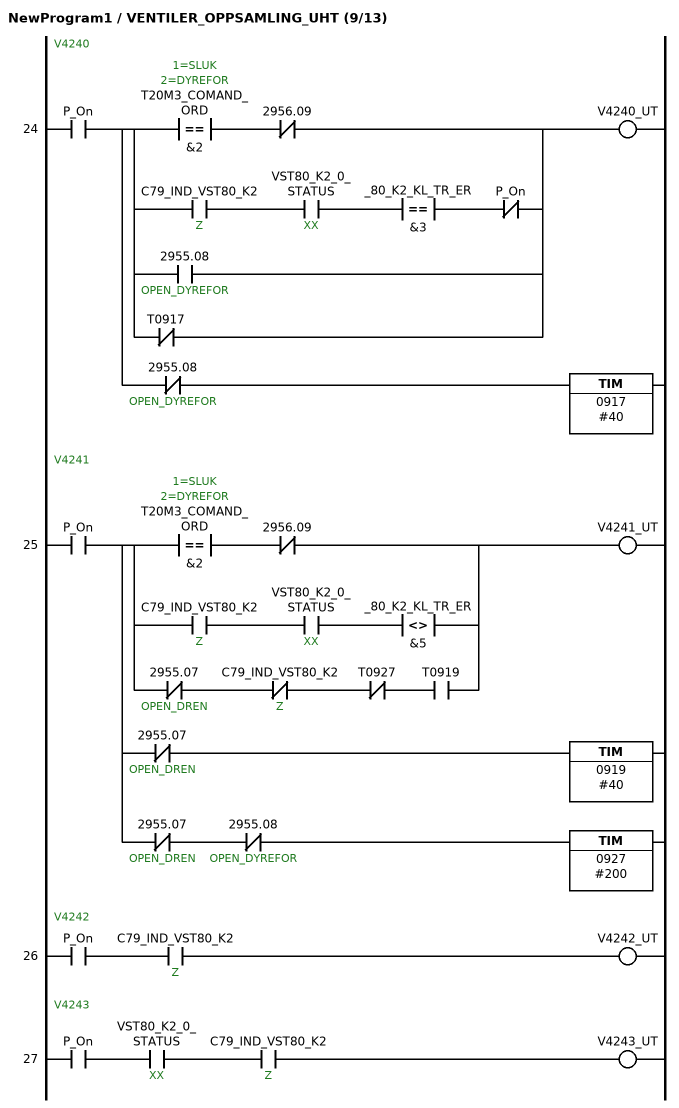
; [picture p888: NewProgram1 / VENTILER_OPPSAMLING_UHT, rungs 24-27]
; rung 24: V4240
LD P_On
OUT TR0
LD=(300) T20M3_COMAND_ORD &2  ; 1=SLUK                                                                     2=DYREFOR
ANDNOT 2956.09
LD C79_IND_VST80_K2  ; Z
AND VST80_K2_0_STATUS  ; XX
AND=(300) _80_K2_KL_TR_ER &3
ANDNOT P_On
ORLD
OR 2955.08  ; OPEN_DYREFOR
ORNOT T0917
ANDLD
OUT V4240_UT
LD TR0
ANDNOT 2955.08  ; OPEN_DYREFOR
TIM 0917 #40
; rung 25: V4241
LD P_On
OUT TR0
LD=(300) T20M3_COMAND_ORD &2  ; 1=SLUK                                                                     2=DYREFOR
ANDNOT 2956.09
LD C79_IND_VST80_K2  ; Z
AND VST80_K2_0_STATUS  ; XX
AND<>(305) _80_K2_KL_TR_ER &5
ORLD
LDNOT 2955.07  ; OPEN_DREN
ANDNOT C79_IND_VST80_K2  ; Z
ANDNOT T0927
AND T0919
ORLD
ANDLD
OUT V4241_UT
LD TR0
ANDNOT 2955.07  ; OPEN_DREN
TIM 0919 #40
LD TR0
ANDNOT 2955.07  ; OPEN_DREN
ANDNOT 2955.08  ; OPEN_DYREFOR
TIM 0927 #200
; rung 26: V4242
LD P_On
AND C79_IND_VST80_K2  ; Z
OUT V4242_UT
; rung 27: V4243
LD P_On
AND VST80_K2_0_STATUS  ; XX
AND C79_IND_VST80_K2  ; Z
OUT V4243_UT

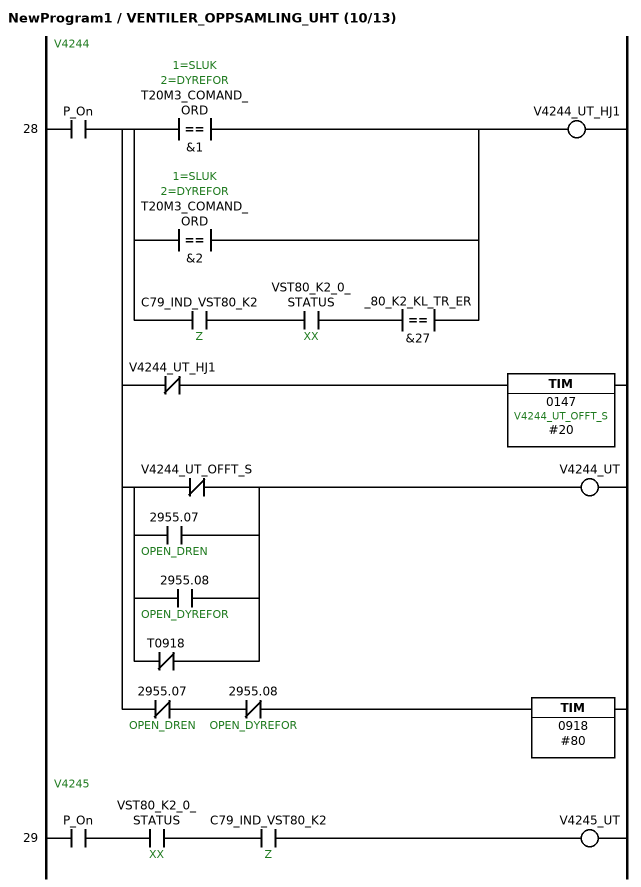
; rung 28: V4244
LD P_On
OUT TR0
LD=(300) T20M3_COMAND_ORD &1  ; 1=SLUK                                                                     2=DYREFOR
OR=(300) T20M3_COMAND_ORD &2  ; 1=SLUK                                                                     2=DYREFOR
LD C79_IND_VST80_K2  ; Z
AND VST80_K2_0_STATUS  ; XX
AND=(300) _80_K2_KL_TR_ER &27
ORLD
ANDLD
OUT V4244_UT_HJ1
LD TR0
ANDNOT V4244_UT_HJ1
TIM 0147 #20  ; V4244_UT_OFFT_S
LD TR0
LDNOT V4244_UT_OFFT_S
OR 2955.07  ; OPEN_DREN
OR 2955.08  ; OPEN_DYREFOR
ORNOT T0918
ANDLD
OUT V4244_UT
LD TR0
ANDNOT 2955.07  ; OPEN_DREN
ANDNOT 2955.08  ; OPEN_DYREFOR
TIM 0918 #80
; rung 29: V4245
LD P_On
AND VST80_K2_0_STATUS  ; XX
AND C79_IND_VST80_K2  ; Z
OUT V4245_UT

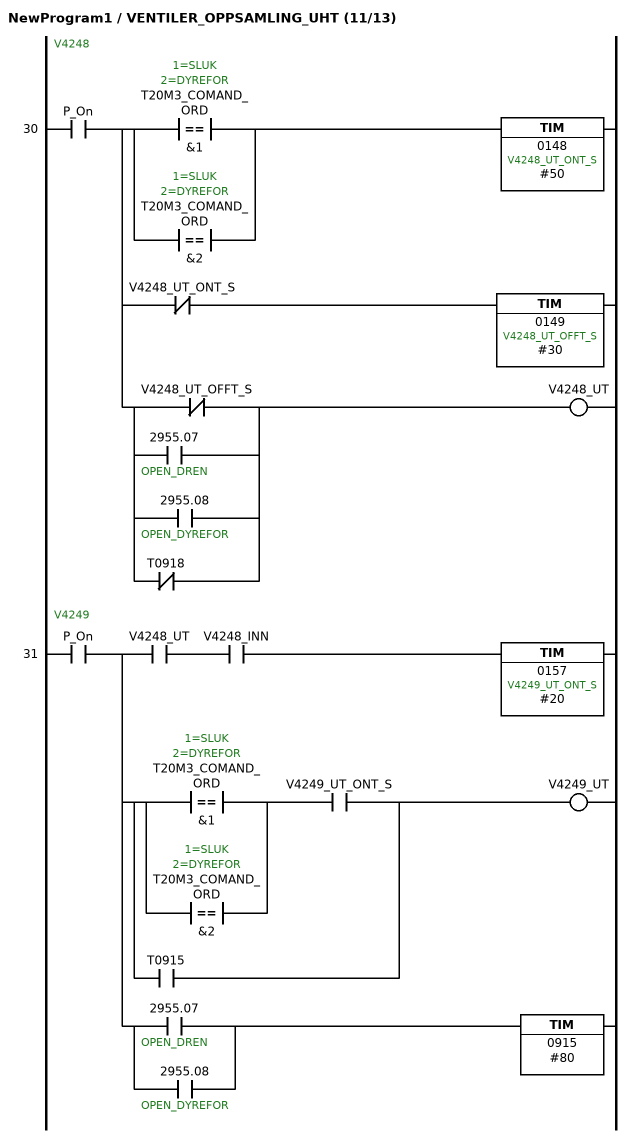
; rung 30: V4248
LD P_On
OUT TR0
LD=(300) T20M3_COMAND_ORD &1  ; 1=SLUK                                                                     2=DYREFOR
OR=(300) T20M3_COMAND_ORD &2  ; 1=SLUK                                                                     2=DYREFOR
ANDLD
TIM 0148 #50  ; V4248_UT_ONT_S
LD TR0
ANDNOT V4248_UT_ONT_S
TIM 0149 #30  ; V4248_UT_OFFT_S
LD TR0
LDNOT V4248_UT_OFFT_S
OR 2955.07  ; OPEN_DREN
OR 2955.08  ; OPEN_DYREFOR
ORNOT T0918
ANDLD
OUT V4248_UT
; rung 31: V4249
LD P_On
OUT TR0
AND V4248_UT
AND V4248_INN
TIM 0157 #20  ; V4249_UT_ONT_S
LD TR0
LD=(300) T20M3_COMAND_ORD &1  ; 1=SLUK                                                                     2=DYREFOR
OR=(300) T20M3_COMAND_ORD &2  ; 1=SLUK                                                                     2=DYREFOR
AND V4249_UT_ONT_S
OR T0915
ANDLD
OUT V4249_UT
LD TR0
LD 2955.07  ; OPEN_DREN
OR 2955.08  ; OPEN_DYREFOR
ANDLD
TIM 0915 #80

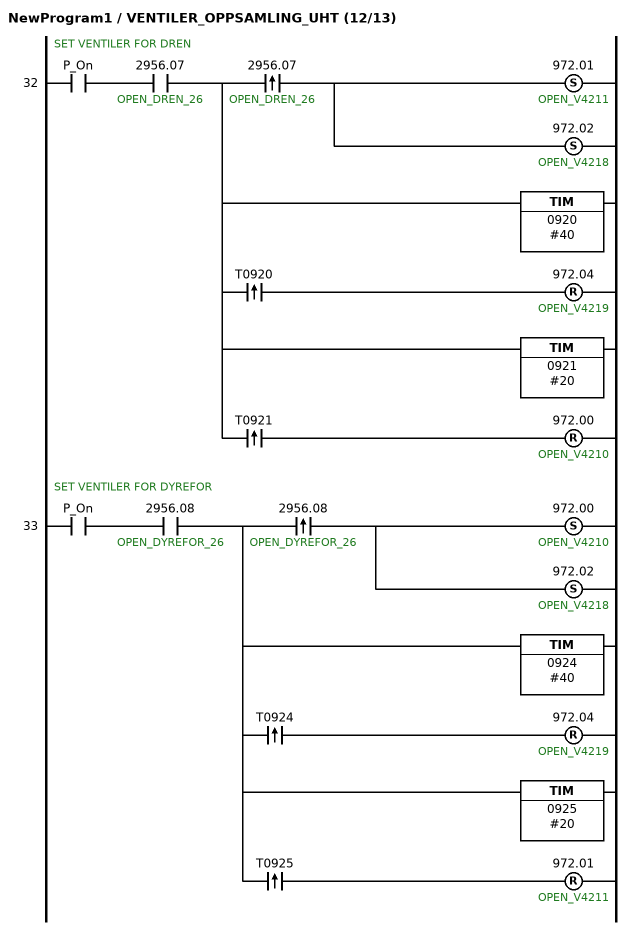
; rung 32: SET VENTILER FOR DREN
LD P_On
AND 2956.07  ; OPEN_DREN_26
OUT TR0
@AND 2956.07  ; OPEN_DREN_26
SET 972.01  ; OPEN_V4211
SET 972.02  ; OPEN_V4218
LD TR0
TIM 0920 #40
@AND T0920
RSET 972.04  ; OPEN_V4219
LD TR0
TIM 0921 #20
@AND T0921
RSET 972.00  ; OPEN_V4210
; rung 33: SET VENTILER FOR DYREFOR
LD P_On
AND 2956.08  ; OPEN_DYREFOR_26
OUT TR0
@AND 2956.08  ; OPEN_DYREFOR_26
SET 972.00  ; OPEN_V4210
SET 972.02  ; OPEN_V4218
LD TR0
TIM 0924 #40
@AND T0924
RSET 972.04  ; OPEN_V4219
LD TR0
TIM 0925 #20
@AND T0925
RSET 972.01  ; OPEN_V4211

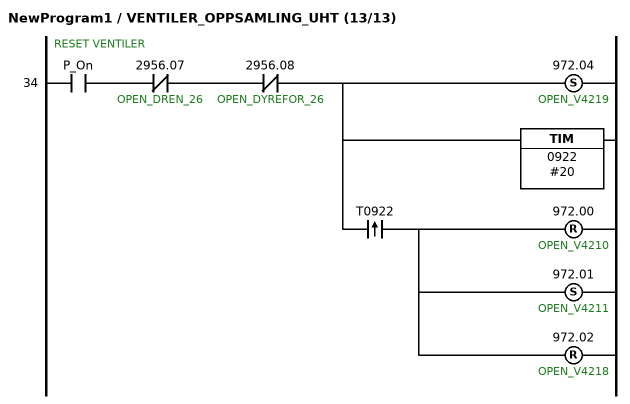
; rung 34: RESET VENTILER
LD P_On
ANDNOT 2956.07  ; OPEN_DREN_26
ANDNOT 2956.08  ; OPEN_DYREFOR_26
SET 972.04  ; OPEN_V4219
TIM 0922 #20
@AND T0922
RSET 972.00  ; OPEN_V4210
SET 972.01  ; OPEN_V4211
RSET 972.02  ; OPEN_V4218
; rung 35: Ingen_kommentar_funnet

### Section PUMPER_SILO_PASTEURER

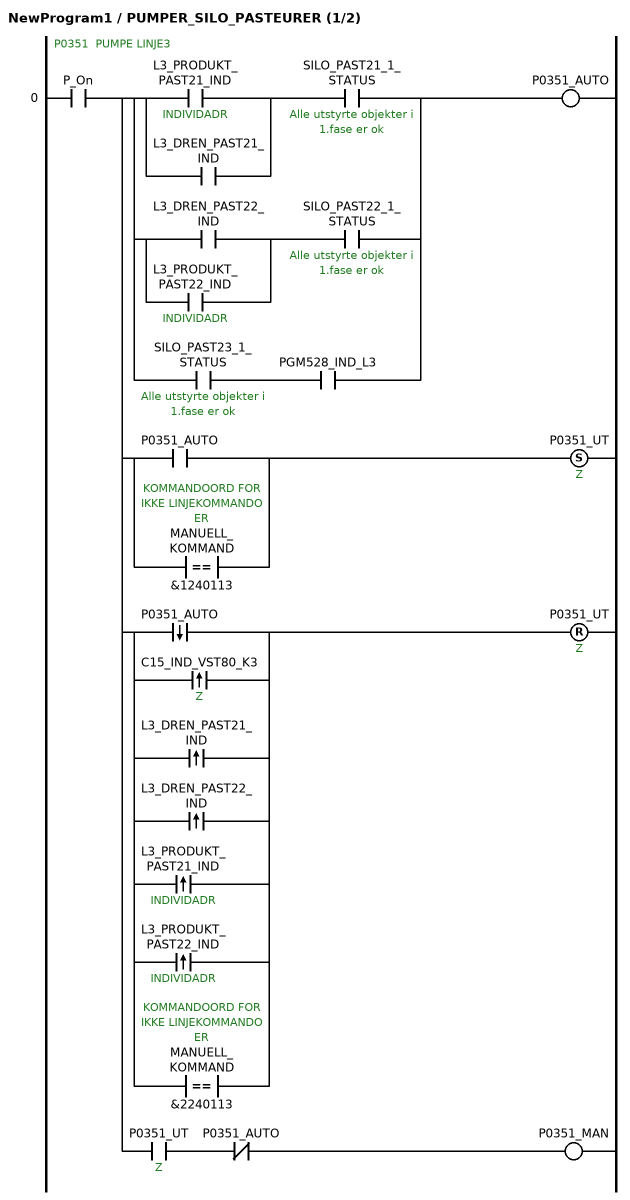
; rung 0: P0351  PUMPE LINJE3
LD P_On
OUT TR0
LD L3_PRODUKT_PAST21_IND  ; INDIVIDADR
OR L3_DREN_PAST21_IND
AND SILO_PAST21_1_STATUS  ; Alle utstyrte objekter i 1.fase er ok
LD L3_DREN_PAST22_IND
OR L3_PRODUKT_PAST22_IND  ; INDIVIDADR
AND SILO_PAST22_1_STATUS  ; Alle utstyrte objekter i 1.fase er ok
ORLD
LD SILO_PAST23_1_STATUS  ; Alle utstyrte objekter i 1.fase er ok
AND PGM528_IND_L3
ORLD
ANDLD
OUT P0351_AUTO
LD TR0
LD P0351_AUTO
OR=L(301) MANUELL_KOMMAND &1240113  ; KOMMANDOORD FOR IKKE LINJEKOMMANDOER
ANDLD
SET P0351_UT  ; Z
LD TR0
%LD P0351_AUTO
@OR C15_IND_VST80_K3  ; Z
@OR L3_DREN_PAST21_IND
@OR L3_DREN_PAST22_IND
@OR L3_PRODUKT_PAST21_IND  ; INDIVIDADR
@OR L3_PRODUKT_PAST22_IND  ; INDIVIDADR
OR=L(301) MANUELL_KOMMAND &2240113  ; KOMMANDOORD FOR IKKE LINJEKOMMANDOER
ANDLD
RSET P0351_UT  ; Z
LD TR0
AND P0351_UT  ; Z
ANDNOT P0351_AUTO
OUT P0351_MAN

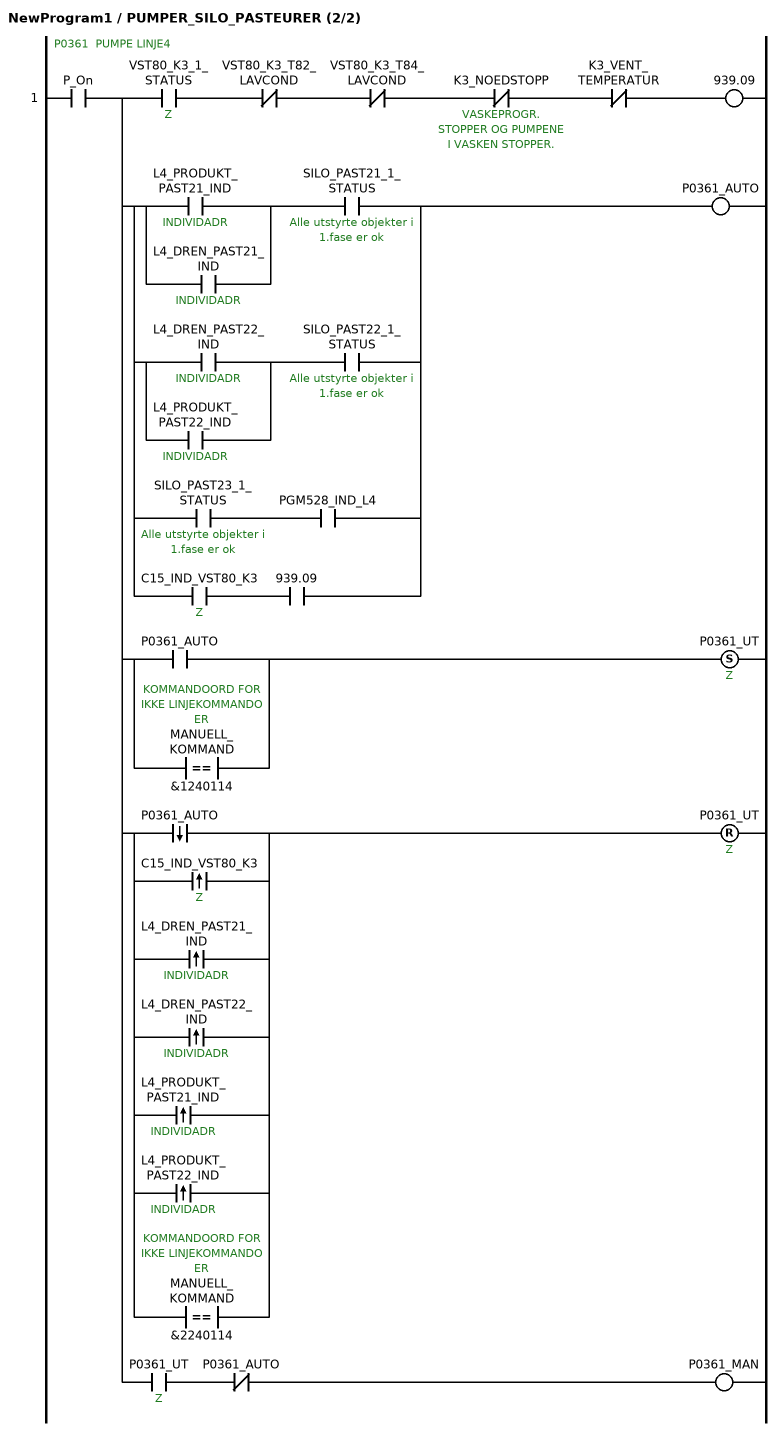
; rung 1: P0361  PUMPE LINJE4
LD P_On
OUT TR0
AND VST80_K3_1_STATUS  ; Z
ANDNOT VST80_K3_T82_LAVCOND
ANDNOT VST80_K3_T84_LAVCOND
ANDNOT K3_NOEDSTOPP  ; VASKEPROGR. STOPPER OG PUMPENE I VASKEN STOPPER.
ANDNOT K3_VENT_TEMPERATUR
OUT 939.09
LD TR0
LD L4_PRODUKT_PAST21_IND  ; INDIVIDADR
OR L4_DREN_PAST21_IND  ; INDIVIDADR
AND SILO_PAST21_1_STATUS  ; Alle utstyrte objekter i 1.fase er ok
LD L4_DREN_PAST22_IND  ; INDIVIDADR
OR L4_PRODUKT_PAST22_IND  ; INDIVIDADR
AND SILO_PAST22_1_STATUS  ; Alle utstyrte objekter i 1.fase er ok
ORLD
LD SILO_PAST23_1_STATUS  ; Alle utstyrte objekter i 1.fase er ok
AND PGM528_IND_L4
ORLD
LD C15_IND_VST80_K3  ; Z
AND 939.09
ORLD
ANDLD
OUT P0361_AUTO
LD TR0
LD P0361_AUTO
OR=L(301) MANUELL_KOMMAND &1240114  ; KOMMANDOORD FOR IKKE LINJEKOMMANDOER
ANDLD
SET P0361_UT  ; Z
LD TR0
%LD P0361_AUTO
@OR C15_IND_VST80_K3  ; Z
@OR L4_DREN_PAST21_IND  ; INDIVIDADR
@OR L4_DREN_PAST22_IND  ; INDIVIDADR
@OR L4_PRODUKT_PAST21_IND  ; INDIVIDADR
@OR L4_PRODUKT_PAST22_IND  ; INDIVIDADR
OR=L(301) MANUELL_KOMMAND &2240114  ; KOMMANDOORD FOR IKKE LINJEKOMMANDOER
ANDLD
RSET P0361_UT  ; Z
LD TR0
AND P0361_UT  ; Z
ANDNOT P0361_AUTO
OUT P0361_MAN
; rung 2: Ingen_kommentar_funnet

### Section MANUELL_OVERPUMPING_SILO

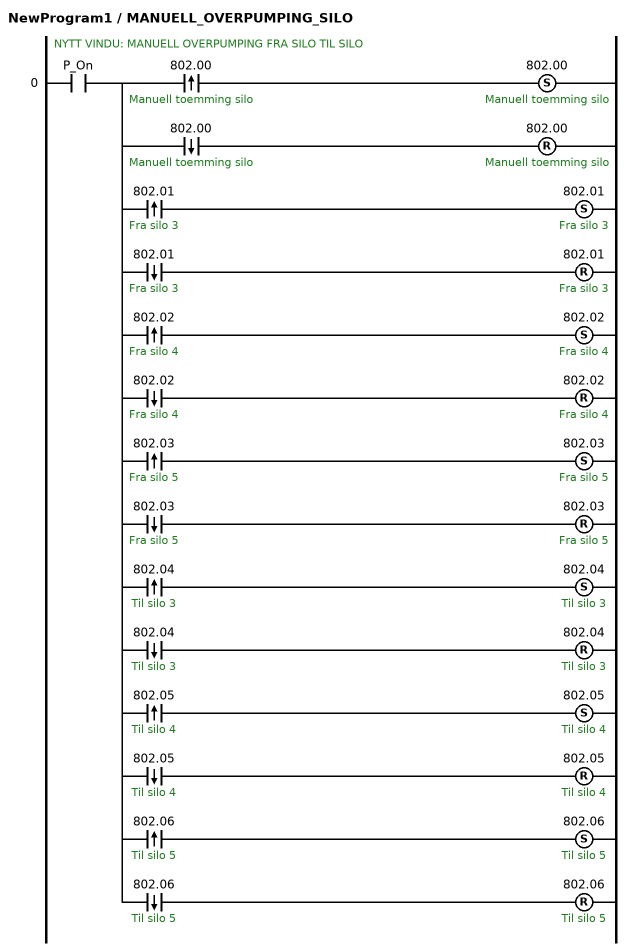
; rung 0: NYTT VINDU: MANUELL OVERPUMPING FRA SILO TIL SILO
LD P_On
OUT TR0
@AND 802.00  ; Manuell toemming silo
SET 802.00  ; Manuell toemming silo
LD TR0
%AND 802.00  ; Manuell toemming silo
RSET 802.00  ; Manuell toemming silo
LD TR0
@AND 802.01  ; Fra silo 3
SET 802.01  ; Fra silo 3
LD TR0
%AND 802.01  ; Fra silo 3
RSET 802.01  ; Fra silo 3
LD TR0
@AND 802.02  ; Fra silo 4
SET 802.02  ; Fra silo 4
LD TR0
%AND 802.02  ; Fra silo 4
RSET 802.02  ; Fra silo 4
LD TR0
@AND 802.03  ; Fra silo 5
SET 802.03  ; Fra silo 5
LD TR0
%AND 802.03  ; Fra silo 5
RSET 802.03  ; Fra silo 5
LD TR0
@AND 802.04  ; Til silo 3
SET 802.04  ; Til silo 3
LD TR0
%AND 802.04  ; Til silo 3
RSET 802.04  ; Til silo 3
LD TR0
@AND 802.05  ; Til silo 4
SET 802.05  ; Til silo 4
LD TR0
%AND 802.05  ; Til silo 4
RSET 802.05  ; Til silo 4
LD TR0
@AND 802.06  ; Til silo 5
SET 802.06  ; Til silo 5
LD TR0
%AND 802.06  ; Til silo 5
RSET 802.06  ; Til silo 5
; rung 1: Ingen_kommentar_funnet

### Section T03_LOKALDREN

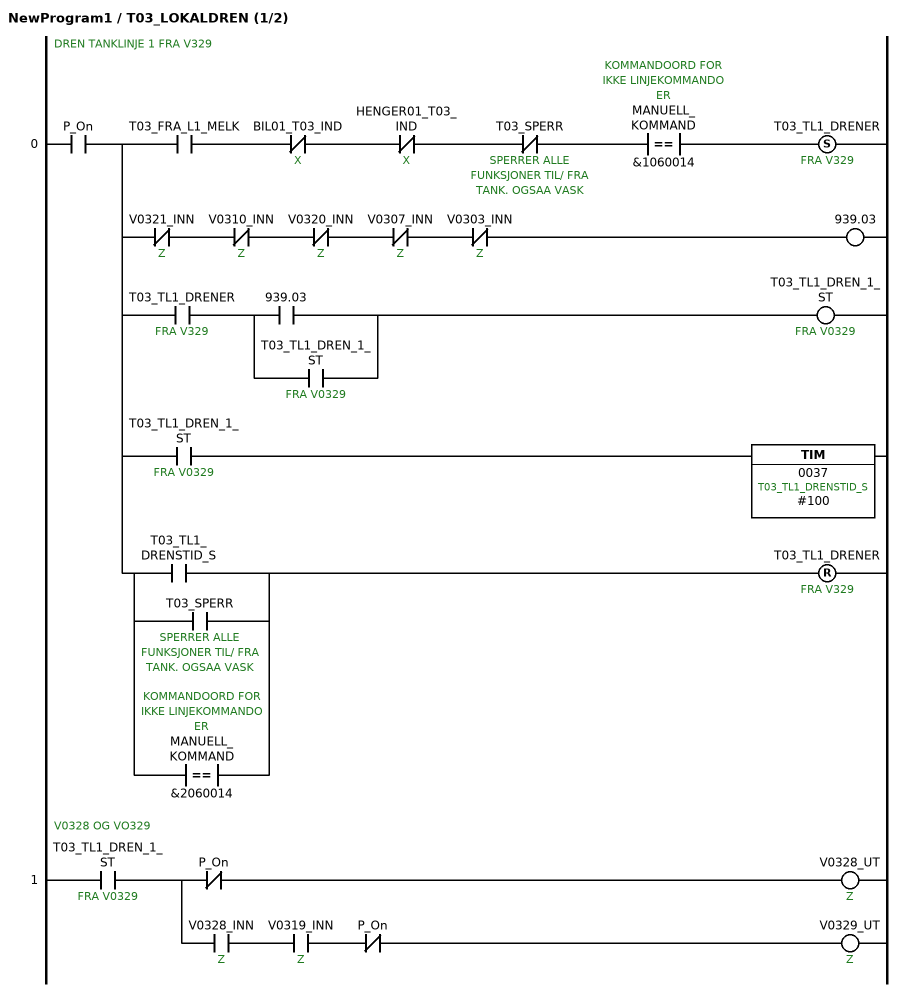
; rung 0: DREN TANKLINJE 1 FRA V329
LD P_On
OUT TR0
AND T03_FRA_L1_MELK
ANDNOT BIL01_T03_IND  ; X
ANDNOT HENGER01_T03_IND  ; X
ANDNOT T03_SPERR  ; SPERRER ALLE FUNKSJONER TIL/ FRA TANK. OGSAA VASK
AND=L(301) MANUELL_KOMMAND &1060014  ; KOMMANDOORD FOR IKKE LINJEKOMMANDOER
SET T03_TL1_DRENER  ; FRA V329
LD TR0
ANDNOT V0321_INN  ; Z
ANDNOT V0310_INN  ; Z
ANDNOT V0320_INN  ; Z
ANDNOT V0307_INN  ; Z
ANDNOT V0303_INN  ; Z
OUT 939.03
LD TR0
AND T03_TL1_DRENER  ; FRA V329
LD 939.03
OR T03_TL1_DREN_1_ST  ; FRA V0329
ANDLD
OUT T03_TL1_DREN_1_ST  ; FRA V0329
LD TR0
AND T03_TL1_DREN_1_ST  ; FRA V0329
TIM 0037 #100  ; T03_TL1_DRENSTID_S
LD TR0
LD T03_TL1_DRENSTID_S
OR T03_SPERR  ; SPERRER ALLE FUNKSJONER TIL/ FRA TANK. OGSAA VASK
OR=L(301) MANUELL_KOMMAND &2060014  ; KOMMANDOORD FOR IKKE LINJEKOMMANDOER
ANDLD
RSET T03_TL1_DRENER  ; FRA V329
; rung 1: V0328 OG VO329
LD T03_TL1_DREN_1_ST  ; FRA V0329
OUT TR0
ANDNOT P_On
OUT V0328_UT  ; Z
LD TR0
AND V0328_INN  ; Z
AND V0319_INN  ; Z
ANDNOT P_On
OUT V0329_UT  ; Z

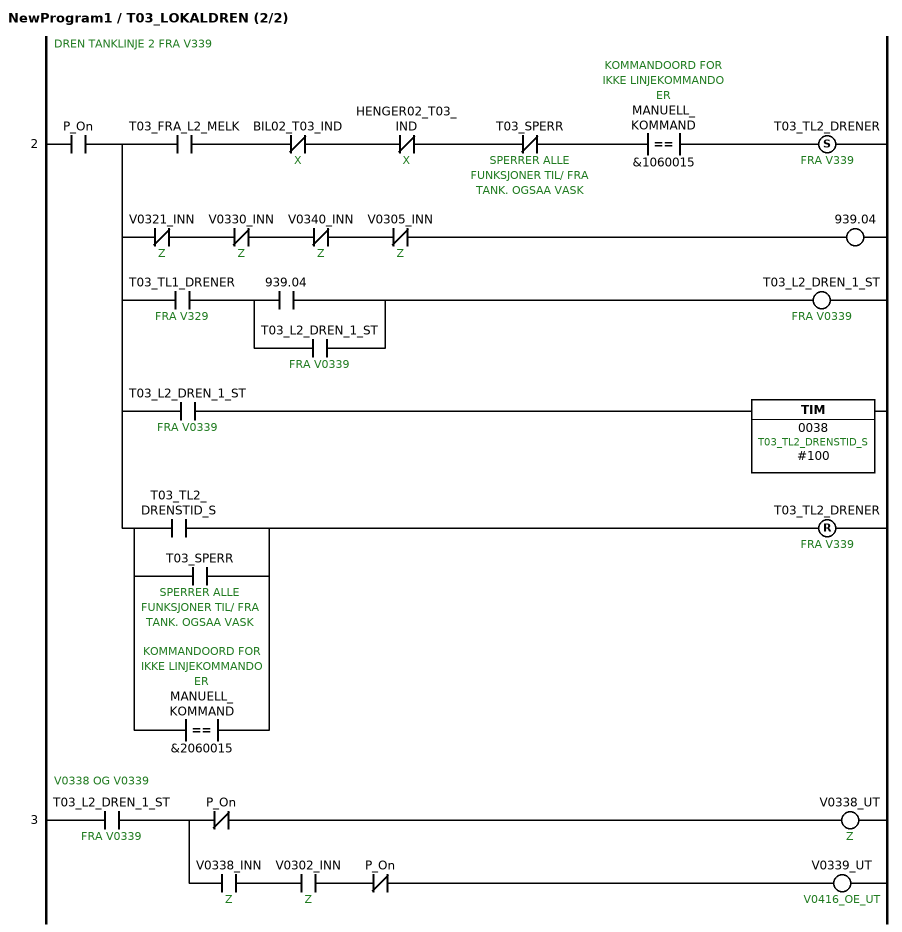
; rung 2: DREN TANKLINJE 2 FRA V339
LD P_On
OUT TR0
AND T03_FRA_L2_MELK
ANDNOT BIL02_T03_IND  ; X
ANDNOT HENGER02_T03_IND  ; X
ANDNOT T03_SPERR  ; SPERRER ALLE FUNKSJONER TIL/ FRA TANK. OGSAA VASK
AND=L(301) MANUELL_KOMMAND &1060015  ; KOMMANDOORD FOR IKKE LINJEKOMMANDOER
SET T03_TL2_DRENER  ; FRA V339
LD TR0
ANDNOT V0321_INN  ; Z
ANDNOT V0330_INN  ; Z
ANDNOT V0340_INN  ; Z
ANDNOT V0305_INN  ; Z
OUT 939.04
LD TR0
AND T03_TL1_DRENER  ; FRA V329
LD 939.04
OR T03_L2_DREN_1_ST  ; FRA V0339
ANDLD
OUT T03_L2_DREN_1_ST  ; FRA V0339
LD TR0
AND T03_L2_DREN_1_ST  ; FRA V0339
TIM 0038 #100  ; T03_TL2_DRENSTID_S
LD TR0
LD T03_TL2_DRENSTID_S
OR T03_SPERR  ; SPERRER ALLE FUNKSJONER TIL/ FRA TANK. OGSAA VASK
OR=L(301) MANUELL_KOMMAND &2060015  ; KOMMANDOORD FOR IKKE LINJEKOMMANDOER
ANDLD
RSET T03_TL2_DRENER  ; FRA V339
; rung 3: V0338 OG V0339
LD T03_L2_DREN_1_ST  ; FRA V0339
OUT TR0
ANDNOT P_On
OUT V0338_UT  ; Z
LD TR0
AND V0338_INN  ; Z
AND V0302_INN  ; Z
ANDNOT P_On
OUT V0339_UT  ; V0416_OE_UT
; rung 4: Ingen_kommentar_funnet

### Section T03_TEMP_NIVÅ

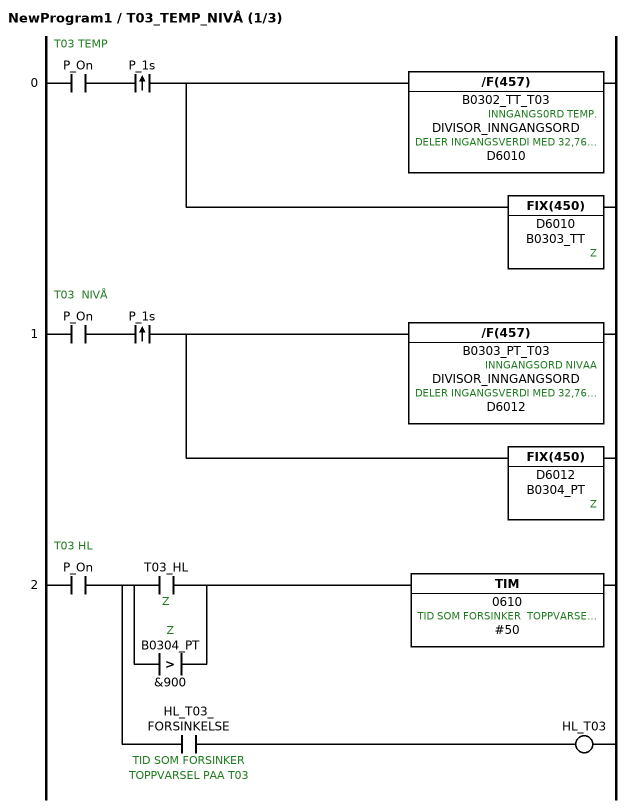
; rung 0: T03 TEMP
LD P_On
@AND P_1s
/F(457) B0302_TT_T03 DIVISOR_INNGANGSORD D6010  ; INNGANGS0RD TEMP., DELER INGANGSVERDI MED 32,760 FOR OMREGNING TIL 0-1000
FIX(450) D6010 B0303_TT  ; Z
; rung 1: T03  NIVÅ
LD P_On
@AND P_1s
/F(457) B0303_PT_T03 DIVISOR_INNGANGSORD D6012  ; INNGANGSORD NIVAA, DELER INGANGSVERDI MED 32,760 FOR OMREGNING TIL 0-1000
FIX(450) D6012 B0304_PT  ; Z
; rung 2: T03 HL
LD P_On
OUT TR0
LD T03_HL  ; Z
OR>(320) B0304_PT &900  ; Z
ANDLD
TIM 0610 #50  ; TID SOM FORSINKER  TOPPVARSEL PAA T03
LD TR0
AND HL_T03_FORSINKELSE  ; TID SOM FORSINKER  TOPPVARSEL PAA T03
OUT HL_T03

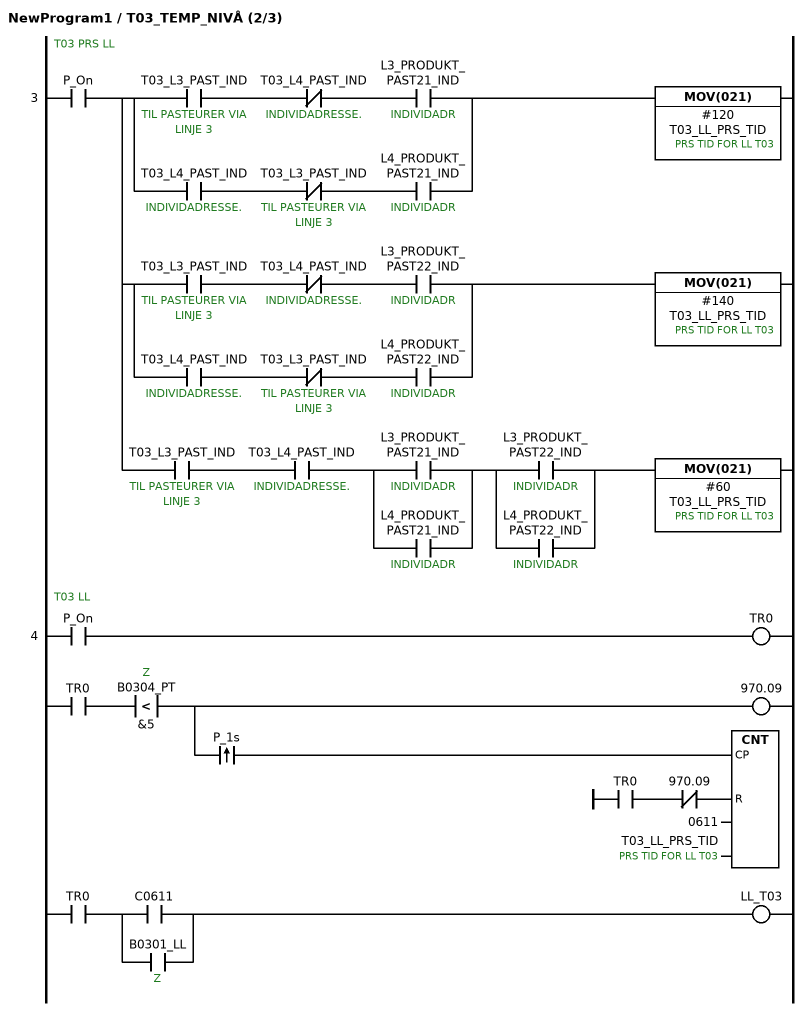
; rung 3: T03 PRS LL
LD P_On
OUT TR0
LD T03_L3_PAST_IND  ; TIL PASTEURER VIA LINJE 3
ANDNOT T03_L4_PAST_IND  ; INDIVIDADRESSE.
AND L3_PRODUKT_PAST21_IND  ; INDIVIDADR
LD T03_L4_PAST_IND  ; INDIVIDADRESSE.
ANDNOT T03_L3_PAST_IND  ; TIL PASTEURER VIA LINJE 3
AND L4_PRODUKT_PAST21_IND  ; INDIVIDADR
ORLD
ANDLD
MOV(021) #120 T03_LL_PRS_TID  ; PRS TID FOR LL T03
LD TR0
LD T03_L3_PAST_IND  ; TIL PASTEURER VIA LINJE 3
ANDNOT T03_L4_PAST_IND  ; INDIVIDADRESSE.
AND L3_PRODUKT_PAST22_IND  ; INDIVIDADR
LD T03_L4_PAST_IND  ; INDIVIDADRESSE.
ANDNOT T03_L3_PAST_IND  ; TIL PASTEURER VIA LINJE 3
AND L4_PRODUKT_PAST22_IND  ; INDIVIDADR
ORLD
ANDLD
MOV(021) #140 T03_LL_PRS_TID  ; PRS TID FOR LL T03
LD TR0
AND T03_L3_PAST_IND  ; TIL PASTEURER VIA LINJE 3
AND T03_L4_PAST_IND  ; INDIVIDADRESSE.
LD L3_PRODUKT_PAST21_IND  ; INDIVIDADR
OR L4_PRODUKT_PAST21_IND  ; INDIVIDADR
ANDLD
LD L3_PRODUKT_PAST22_IND  ; INDIVIDADR
OR L4_PRODUKT_PAST22_IND  ; INDIVIDADR
ANDLD
MOV(021) #60 T03_LL_PRS_TID  ; PRS TID FOR LL T03
; rung 4: T03 LL
LD P_On
OUT TR0
AND<(310) B0304_PT &5  ; Z
OUT 970.09
@AND P_1s
LD TR0
ANDNOT 970.09
CNT 0611 T03_LL_PRS_TID  ; PRS TID FOR LL T03
LD TR0
LD C0611
OR B0301_LL  ; Z
ANDLD
OUT LL_T03

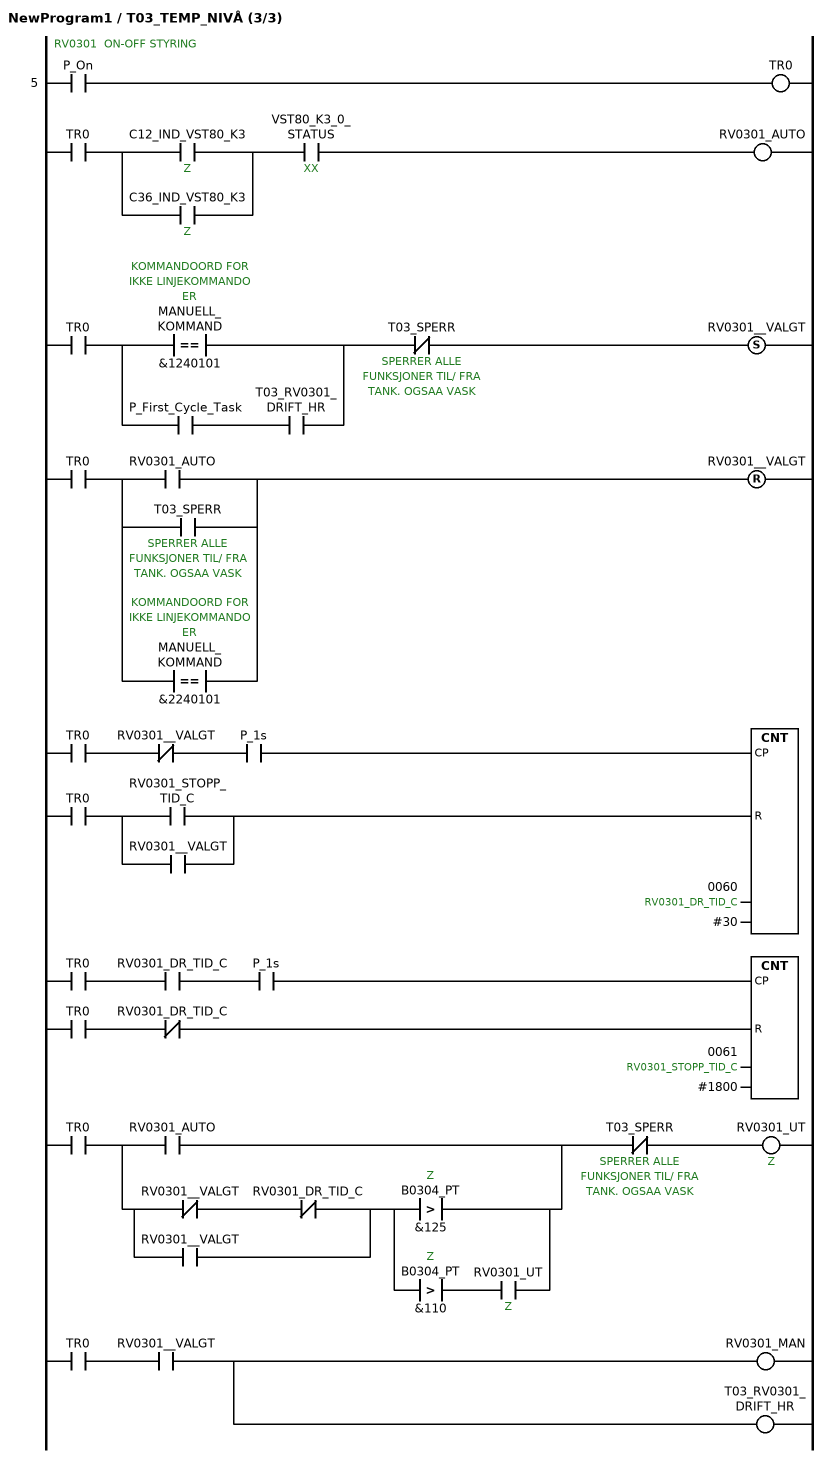
; rung 5: RV0301  ON-OFF STYRING
LD P_On
OUT TR0
LD C12_IND_VST80_K3  ; Z
OR C36_IND_VST80_K3  ; Z
ANDLD
AND VST80_K3_0_STATUS  ; XX
OUT RV0301_AUTO
LD TR0
LD=L(301) MANUELL_KOMMAND &1240101  ; KOMMANDOORD FOR IKKE LINJEKOMMANDOER
LD P_First_Cycle_Task
AND T03_RV0301_DRIFT_HR
ORLD
ANDLD
ANDNOT T03_SPERR  ; SPERRER ALLE FUNKSJONER TIL/ FRA TANK. OGSAA VASK
SET RV0301__VALGT
LD TR0
LD RV0301_AUTO
OR T03_SPERR  ; SPERRER ALLE FUNKSJONER TIL/ FRA TANK. OGSAA VASK
OR=L(301) MANUELL_KOMMAND &2240101  ; KOMMANDOORD FOR IKKE LINJEKOMMANDOER
ANDLD
RSET RV0301__VALGT
LD TR0
ANDNOT RV0301__VALGT
AND P_1s
LD TR0
LD RV0301_STOPP_TID_C
OR RV0301__VALGT
ANDLD
CNT 0060 #30  ; RV0301_DR_TID_C
LD TR0
AND RV0301_DR_TID_C
AND P_1s
LD TR0
ANDNOT RV0301_DR_TID_C
CNT 0061 #1800  ; RV0301_STOPP_TID_C
LD TR0
LD RV0301_AUTO
LDNOT RV0301__VALGT
ANDNOT RV0301_DR_TID_C
OR RV0301__VALGT
LD>(320) B0304_PT &125  ; Z
LD>(320) B0304_PT &110  ; Z
AND RV0301_UT  ; Z
ORLD
ANDLD
ORLD
ANDLD
ANDNOT T03_SPERR  ; SPERRER ALLE FUNKSJONER TIL/ FRA TANK. OGSAA VASK
OUT RV0301_UT  ; Z
LD TR0
AND RV0301__VALGT
OUT RV0301_MAN
OUT T03_RV0301_DRIFT_HR
; rung 6: Ingen_kommentar_funnet

### Section T03_STATUS

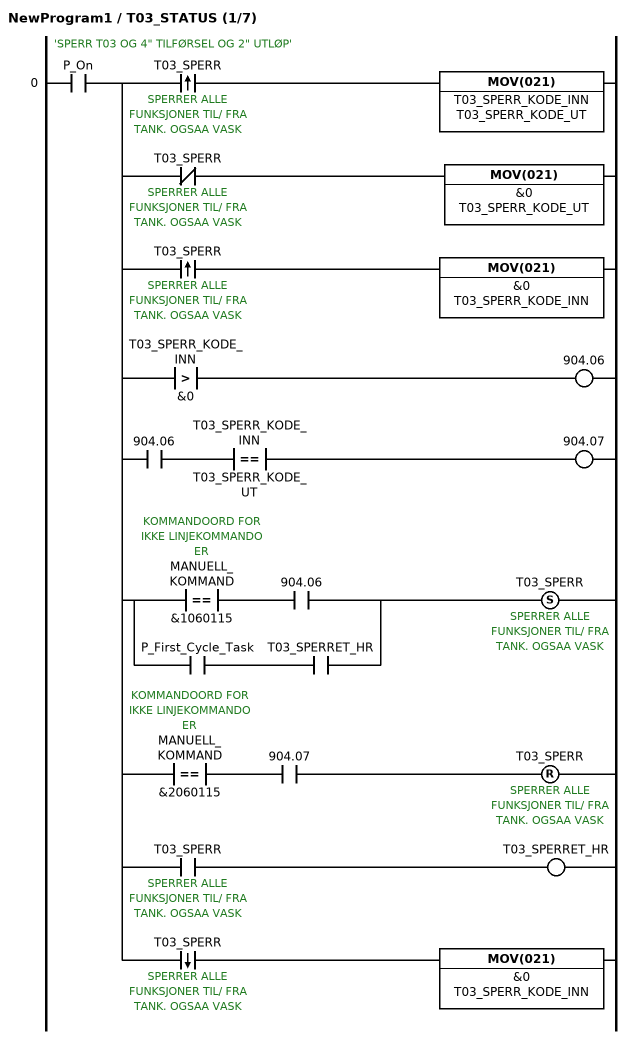
; rung 0: 'SPERR T03 OG 4" TILFØRSEL OG 2" UTLØP'
LD P_On
OUT TR0
@AND T03_SPERR  ; SPERRER ALLE FUNKSJONER TIL/ FRA TANK. OGSAA VASK
MOV(021) T03_SPERR_KODE_INN T03_SPERR_KODE_UT
LD TR0
ANDNOT T03_SPERR  ; SPERRER ALLE FUNKSJONER TIL/ FRA TANK. OGSAA VASK
MOV(021) &0 T03_SPERR_KODE_UT
LD TR0
@AND T03_SPERR  ; SPERRER ALLE FUNKSJONER TIL/ FRA TANK. OGSAA VASK
MOV(021) &0 T03_SPERR_KODE_INN
LD TR0
AND>(320) T03_SPERR_KODE_INN &0
OUT 904.06
LD TR0
AND 904.06
AND=(300) T03_SPERR_KODE_INN T03_SPERR_KODE_UT
OUT 904.07
LD TR0
LD=L(301) MANUELL_KOMMAND &1060115  ; KOMMANDOORD FOR IKKE LINJEKOMMANDOER
AND 904.06
LD P_First_Cycle_Task
AND T03_SPERRET_HR
ORLD
ANDLD
SET T03_SPERR  ; SPERRER ALLE FUNKSJONER TIL/ FRA TANK. OGSAA VASK
LD TR0
AND=L(301) MANUELL_KOMMAND &2060115  ; KOMMANDOORD FOR IKKE LINJEKOMMANDOER
AND 904.07
RSET T03_SPERR  ; SPERRER ALLE FUNKSJONER TIL/ FRA TANK. OGSAA VASK
LD TR0
AND T03_SPERR  ; SPERRER ALLE FUNKSJONER TIL/ FRA TANK. OGSAA VASK
OUT T03_SPERRET_HR
LD TR0
%AND T03_SPERR  ; SPERRER ALLE FUNKSJONER TIL/ FRA TANK. OGSAA VASK
MOV(021) &0 T03_SPERR_KODE_INN

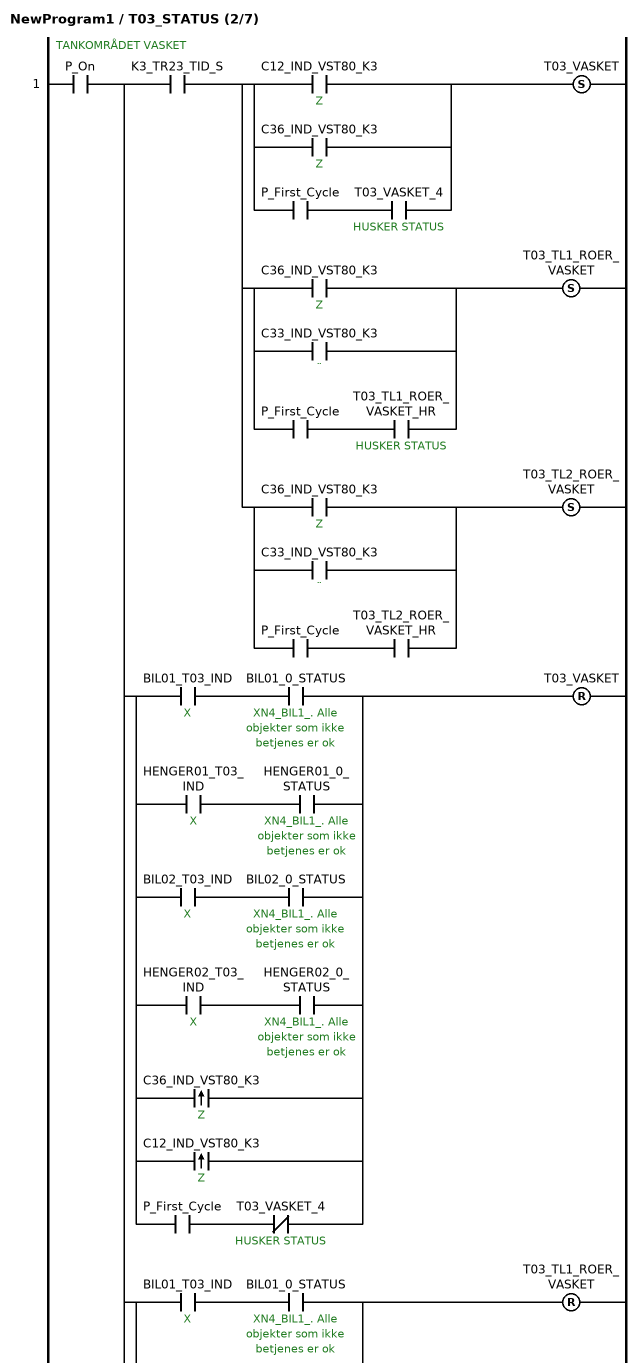

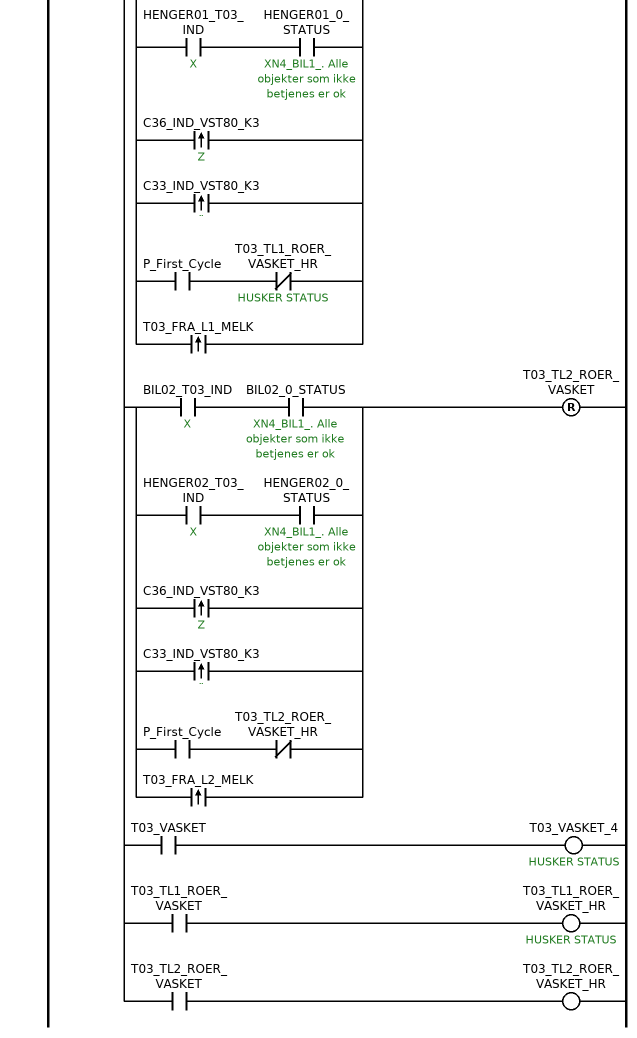
; rung 1: TANKOMRÅDET VASKET
LD P_On
OUT TR0
AND K3_TR23_TID_S
OUT TR1
LD C12_IND_VST80_K3  ; Z
OR C36_IND_VST80_K3  ; Z
LD P_First_Cycle
AND T03_VASKET_4  ; HUSKER STATUS
ORLD
ANDLD
SET T03_VASKET
LD TR1
LD C36_IND_VST80_K3  ; Z
OR C33_IND_VST80_K3  ; ¨
LD P_First_Cycle
AND T03_TL1_ROER_VASKET_HR  ; HUSKER STATUS
ORLD
ANDLD
SET T03_TL1_ROER_VASKET
LD TR1
LD C36_IND_VST80_K3  ; Z
OR C33_IND_VST80_K3  ; ¨
LD P_First_Cycle
AND T03_TL2_ROER_VASKET_HR
ORLD
ANDLD
SET T03_TL2_ROER_VASKET
LD TR0
LD BIL01_T03_IND  ; X
AND BIL01_0_STATUS  ; XN4_BIL1_. Alle objekter som ikke betjenes er ok
LD HENGER01_T03_IND  ; X
AND HENGER01_0_STATUS  ; XN4_BIL1_. Alle objekter som ikke betjenes er ok
ORLD
LD BIL02_T03_IND  ; X
AND BIL02_0_STATUS  ; XN4_BIL1_. Alle objekter som ikke betjenes er ok
ORLD
LD HENGER02_T03_IND  ; X
AND HENGER02_0_STATUS  ; XN4_BIL1_. Alle objekter som ikke betjenes er ok
ORLD
@OR C36_IND_VST80_K3  ; Z
@OR C12_IND_VST80_K3  ; Z
LD P_First_Cycle
ANDNOT T03_VASKET_4  ; HUSKER STATUS
ORLD
ANDLD
RSET T03_VASKET
LD TR0
LD BIL01_T03_IND  ; X
AND BIL01_0_STATUS  ; XN4_BIL1_. Alle objekter som ikke betjenes er ok
LD HENGER01_T03_IND  ; X
AND HENGER01_0_STATUS  ; XN4_BIL1_. Alle objekter som ikke betjenes er ok
ORLD
@OR C36_IND_VST80_K3  ; Z
@OR C33_IND_VST80_K3  ; ¨
LD P_First_Cycle
ANDNOT T03_TL1_ROER_VASKET_HR  ; HUSKER STATUS
ORLD
@OR T03_FRA_L1_MELK
ANDLD
RSET T03_TL1_ROER_VASKET
LD TR0
LD BIL02_T03_IND  ; X
AND BIL02_0_STATUS  ; XN4_BIL1_. Alle objekter som ikke betjenes er ok
LD HENGER02_T03_IND  ; X
AND HENGER02_0_STATUS  ; XN4_BIL1_. Alle objekter som ikke betjenes er ok
ORLD
@OR C36_IND_VST80_K3  ; Z
@OR C33_IND_VST80_K3  ; ¨
LD P_First_Cycle
ANDNOT T03_TL2_ROER_VASKET_HR
ORLD
@OR T03_FRA_L2_MELK
ANDLD
RSET T03_TL2_ROER_VASKET
LD TR0
AND T03_VASKET
OUT T03_VASKET_4  ; HUSKER STATUS
LD TR0
AND T03_TL1_ROER_VASKET
OUT T03_TL1_ROER_VASKET_HR  ; HUSKER STATUS
LD TR0
AND T03_TL2_ROER_VASKET
OUT T03_TL2_ROER_VASKET_HR

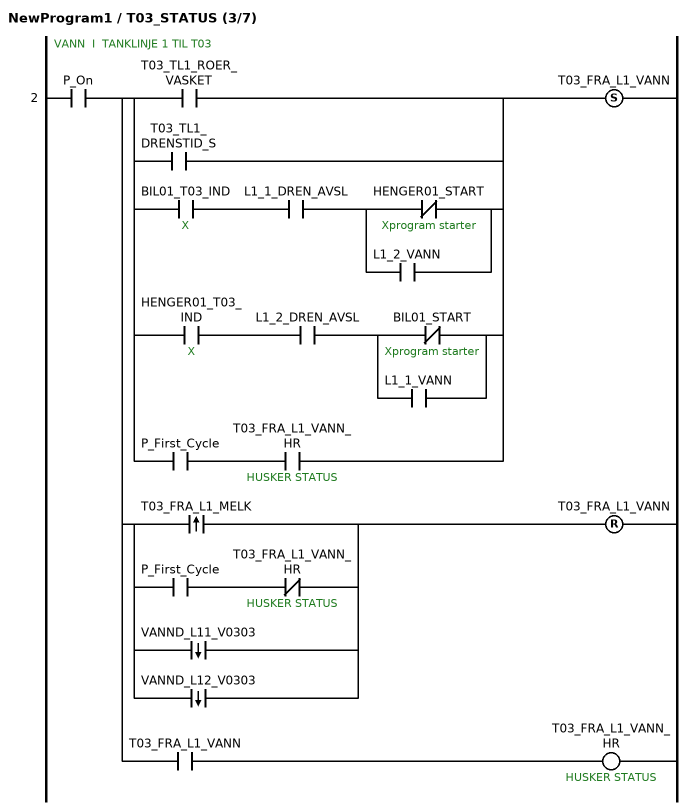
; rung 2: VANN  I  TANKLINJE 1 TIL T03
LD P_On
OUT TR0
LD T03_TL1_ROER_VASKET
OR T03_TL1_DRENSTID_S
LD BIL01_T03_IND  ; X
AND L1_1_DREN_AVSL
LDNOT HENGER01_START  ; Xprogram starter
OR L1_2_VANN
ANDLD
ORLD
LD HENGER01_T03_IND  ; X
AND L1_2_DREN_AVSL
LDNOT BIL01_START  ; Xprogram starter
OR L1_1_VANN
ANDLD
ORLD
LD P_First_Cycle
AND T03_FRA_L1_VANN_HR  ; HUSKER STATUS
ORLD
ANDLD
SET T03_FRA_L1_VANN
LD TR0
@LD T03_FRA_L1_MELK
LD P_First_Cycle
ANDNOT T03_FRA_L1_VANN_HR  ; HUSKER STATUS
ORLD
%OR VANND_L11_V0303
%OR VANND_L12_V0303
ANDLD
RSET T03_FRA_L1_VANN
LD TR0
AND T03_FRA_L1_VANN
OUT T03_FRA_L1_VANN_HR  ; HUSKER STATUS

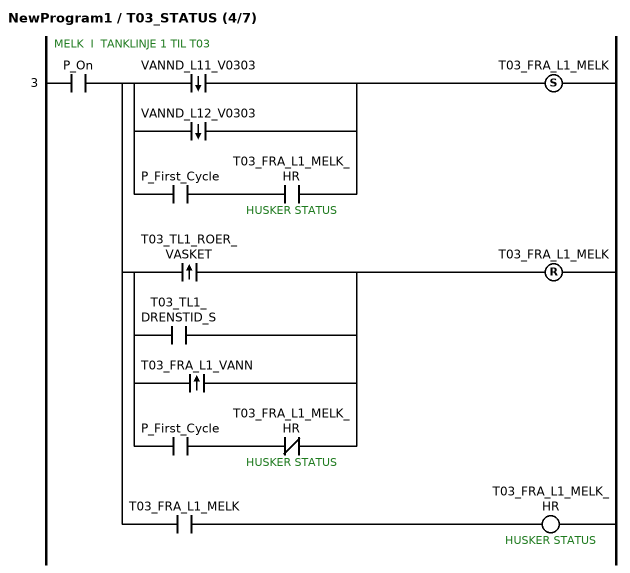
; rung 3: MELK  I  TANKLINJE 1 TIL T03
LD P_On
OUT TR0
%LD VANND_L11_V0303
%OR VANND_L12_V0303
LD P_First_Cycle
AND T03_FRA_L1_MELK_HR  ; HUSKER STATUS
ORLD
ANDLD
SET T03_FRA_L1_MELK
LD TR0
@LD T03_TL1_ROER_VASKET
OR T03_TL1_DRENSTID_S
@OR T03_FRA_L1_VANN
LD P_First_Cycle
ANDNOT T03_FRA_L1_MELK_HR  ; HUSKER STATUS
ORLD
ANDLD
RSET T03_FRA_L1_MELK
LD TR0
AND T03_FRA_L1_MELK
OUT T03_FRA_L1_MELK_HR  ; HUSKER STATUS

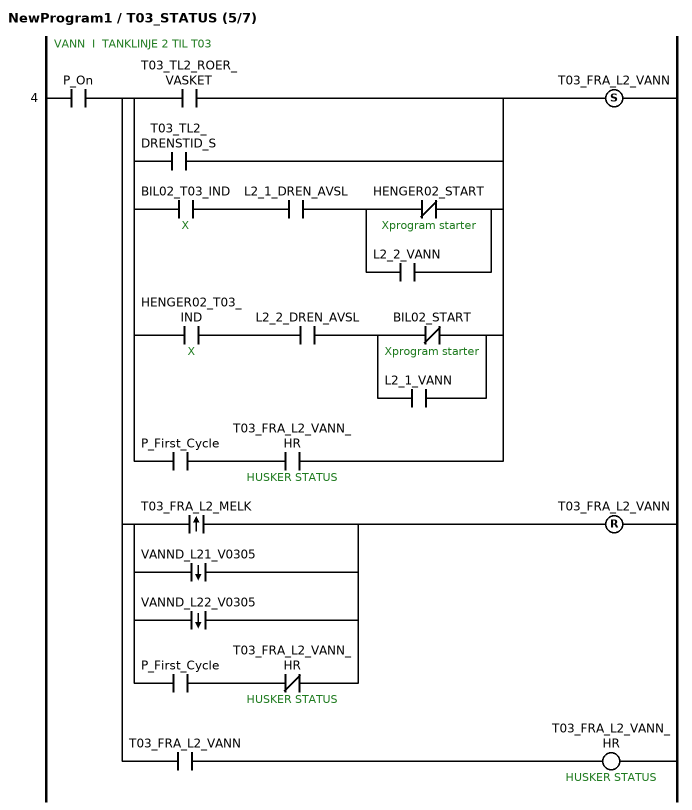
; rung 4: VANN  I  TANKLINJE 2 TIL T03
LD P_On
OUT TR0
LD T03_TL2_ROER_VASKET
OR T03_TL2_DRENSTID_S
LD BIL02_T03_IND  ; X
AND L2_1_DREN_AVSL
LDNOT HENGER02_START  ; Xprogram starter
OR L2_2_VANN
ANDLD
ORLD
LD HENGER02_T03_IND  ; X
AND L2_2_DREN_AVSL
LDNOT BIL02_START  ; Xprogram starter
OR L2_1_VANN
ANDLD
ORLD
LD P_First_Cycle
AND T03_FRA_L2_VANN_HR  ; HUSKER STATUS
ORLD
ANDLD
SET T03_FRA_L2_VANN
LD TR0
@LD T03_FRA_L2_MELK
%OR VANND_L21_V0305
%OR VANND_L22_V0305
LD P_First_Cycle
ANDNOT T03_FRA_L2_VANN_HR  ; HUSKER STATUS
ORLD
ANDLD
RSET T03_FRA_L2_VANN
LD TR0
AND T03_FRA_L2_VANN
OUT T03_FRA_L2_VANN_HR  ; HUSKER STATUS

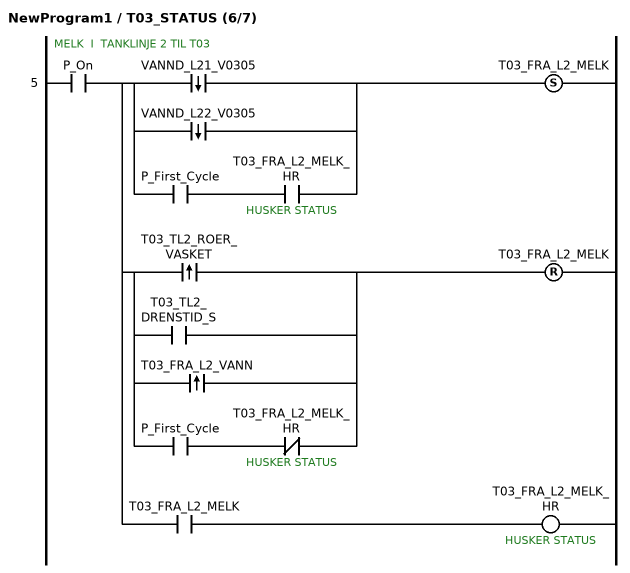
; rung 5: MELK  I  TANKLINJE 2 TIL T03
LD P_On
OUT TR0
%LD VANND_L21_V0305
%OR VANND_L22_V0305
LD P_First_Cycle
AND T03_FRA_L2_MELK_HR  ; HUSKER STATUS
ORLD
ANDLD
SET T03_FRA_L2_MELK
LD TR0
@LD T03_TL2_ROER_VASKET
OR T03_TL2_DRENSTID_S
@OR T03_FRA_L2_VANN
LD P_First_Cycle
ANDNOT T03_FRA_L2_MELK_HR  ; HUSKER STATUS
ORLD
ANDLD
RSET T03_FRA_L2_MELK
LD TR0
AND T03_FRA_L2_MELK
OUT T03_FRA_L2_MELK_HR  ; HUSKER STATUS

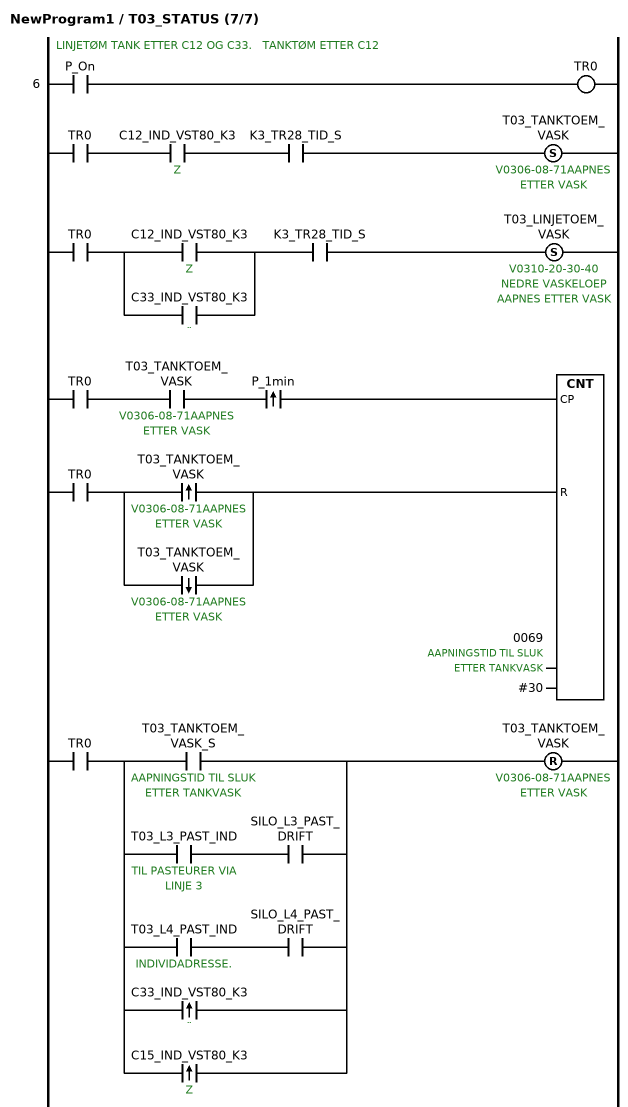

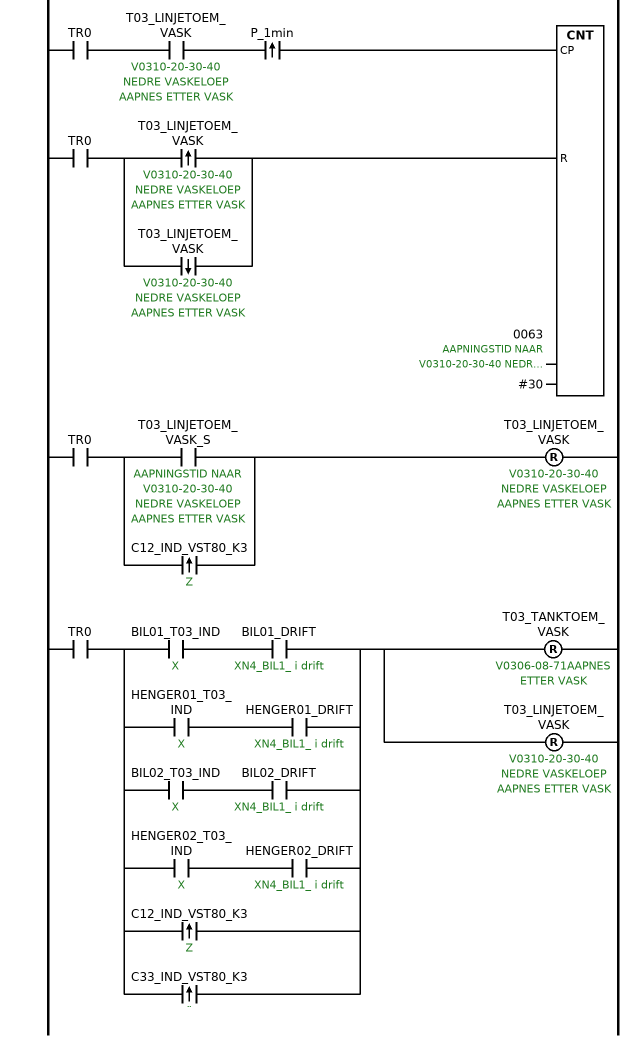
; rung 6: LINJETØM TANK ETTER C12 OG C33.   TANKTØM ETTER C12
LD P_On
OUT TR0
AND C12_IND_VST80_K3  ; Z
AND K3_TR28_TID_S
SET T03_TANKTOEM_VASK  ; V0306-08-71AAPNES ETTER VASK
LD TR0
LD C12_IND_VST80_K3  ; Z
OR C33_IND_VST80_K3  ; ¨
ANDLD
AND K3_TR28_TID_S
SET T03_LINJETOEM_VASK  ; V0310-20-30-40 NEDRE VASKELOEP AAPNES ETTER VASK
LD TR0
AND T03_TANKTOEM_VASK  ; V0306-08-71AAPNES ETTER VASK
@AND P_1min
LD TR0
@LD T03_TANKTOEM_VASK  ; V0306-08-71AAPNES ETTER VASK
%OR T03_TANKTOEM_VASK  ; V0306-08-71AAPNES ETTER VASK
ANDLD
CNT 0069 #30  ; AAPNINGSTID TIL SLUK ETTER TANKVASK
LD TR0
LD T03_TANKTOEM_VASK_S  ; AAPNINGSTID TIL SLUK ETTER TANKVASK
LD T03_L3_PAST_IND  ; TIL PASTEURER VIA LINJE 3
AND SILO_L3_PAST_DRIFT
ORLD
LD T03_L4_PAST_IND  ; INDIVIDADRESSE.
AND SILO_L4_PAST_DRIFT
ORLD
@OR C33_IND_VST80_K3  ; ¨
@OR C15_IND_VST80_K3  ; Z
ANDLD
RSET T03_TANKTOEM_VASK  ; V0306-08-71AAPNES ETTER VASK
LD TR0
AND T03_LINJETOEM_VASK  ; V0310-20-30-40 NEDRE VASKELOEP AAPNES ETTER VASK
@AND P_1min
LD TR0
@LD T03_LINJETOEM_VASK  ; V0310-20-30-40 NEDRE VASKELOEP AAPNES ETTER VASK
%OR T03_LINJETOEM_VASK  ; V0310-20-30-40 NEDRE VASKELOEP AAPNES ETTER VASK
ANDLD
CNT 0063 #30  ; AAPNINGSTID NAAR V0310-20-30-40 NEDRE VASKELOEP AAPNES ETTER VASK
LD TR0
LD T03_LINJETOEM_VASK_S  ; AAPNINGSTID NAAR V0310-20-30-40 NEDRE VASKELOEP AAPNES ETTER VASK
@OR C12_IND_VST80_K3  ; Z
ANDLD
RSET T03_LINJETOEM_VASK  ; V0310-20-30-40 NEDRE VASKELOEP AAPNES ETTER VASK
LD TR0
LD BIL01_T03_IND  ; X
AND BIL01_DRIFT  ; XN4_BIL1_ i drift
LD HENGER01_T03_IND  ; X
AND HENGER01_DRIFT  ; XN4_BIL1_ i drift
ORLD
LD BIL02_T03_IND  ; X
AND BIL02_DRIFT  ; XN4_BIL1_ i drift
ORLD
LD HENGER02_T03_IND  ; X
AND HENGER02_DRIFT  ; XN4_BIL1_ i drift
ORLD
@OR C12_IND_VST80_K3  ; Z
@OR C33_IND_VST80_K3  ; ¨
ANDLD
RSET T03_TANKTOEM_VASK  ; V0306-08-71AAPNES ETTER VASK
RSET T03_LINJETOEM_VASK  ; V0310-20-30-40 NEDRE VASKELOEP AAPNES ETTER VASK
; rung 7: Ingen_kommentar_funnet

### Section T04_LOKALDREN

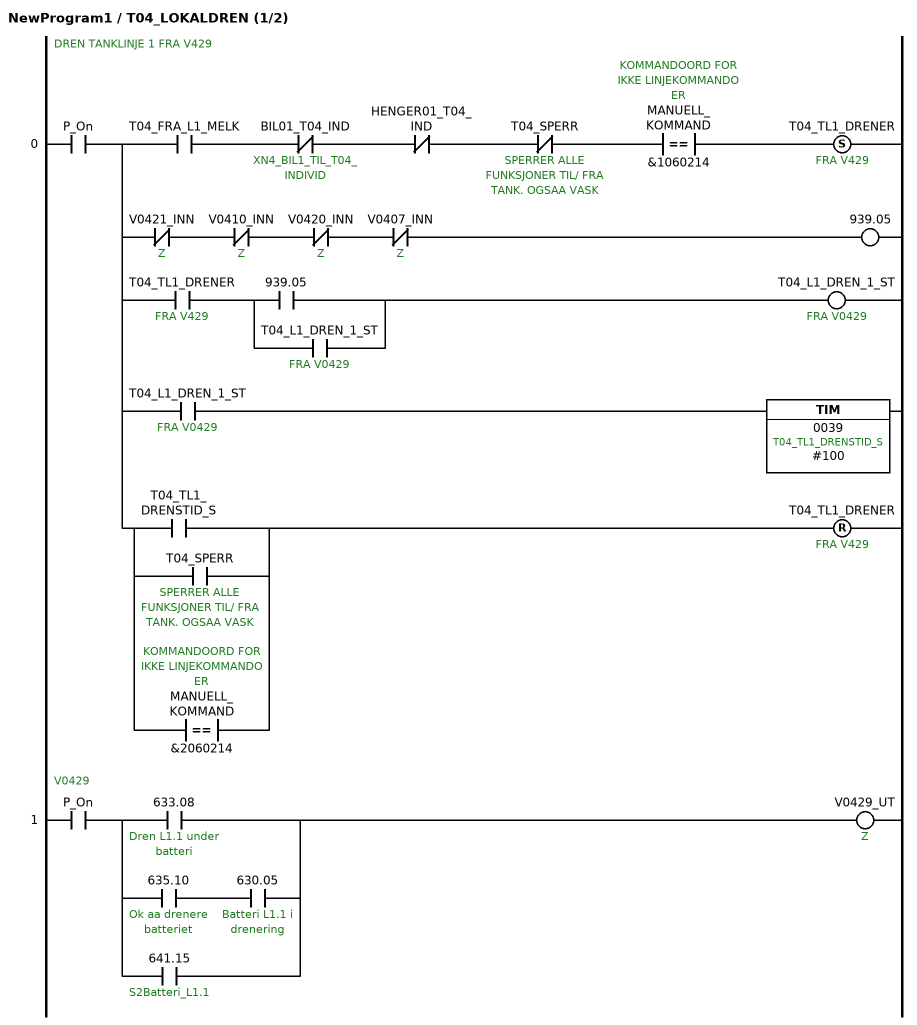
; rung 0: DREN TANKLINJE 1 FRA V429
LD P_On
OUT TR0
AND T04_FRA_L1_MELK
ANDNOT BIL01_T04_IND  ; XN4_BIL1_TIL_T04_INDIVID
ANDNOT HENGER01_T04_IND
ANDNOT T04_SPERR  ; SPERRER ALLE FUNKSJONER TIL/ FRA TANK. OGSAA VASK
AND=L(301) MANUELL_KOMMAND &1060214  ; KOMMANDOORD FOR IKKE LINJEKOMMANDOER
SET T04_TL1_DRENER  ; FRA V429
LD TR0
ANDNOT V0421_INN  ; Z
ANDNOT V0410_INN  ; Z
ANDNOT V0420_INN  ; Z
ANDNOT V0407_INN  ; Z
OUT 939.05
LD TR0
AND T04_TL1_DRENER  ; FRA V429
LD 939.05
OR T04_L1_DREN_1_ST  ; FRA V0429
ANDLD
OUT T04_L1_DREN_1_ST  ; FRA V0429
LD TR0
AND T04_L1_DREN_1_ST  ; FRA V0429
TIM 0039 #100  ; T04_TL1_DRENSTID_S
LD TR0
LD T04_TL1_DRENSTID_S
OR T04_SPERR  ; SPERRER ALLE FUNKSJONER TIL/ FRA TANK. OGSAA VASK
OR=L(301) MANUELL_KOMMAND &2060214  ; KOMMANDOORD FOR IKKE LINJEKOMMANDOER
ANDLD
RSET T04_TL1_DRENER  ; FRA V429
; rung 1: V0429
LD P_On
LD 633.08  ; Dren L1.1 under batteri
LD 635.10  ; Ok aa drenere batteriet
AND 630.05  ; Batteri L1.1 i drenering
ORLD
OR 641.15  ; S2Batteri_L1.1
ANDLD
OUT V0429_UT  ; Z

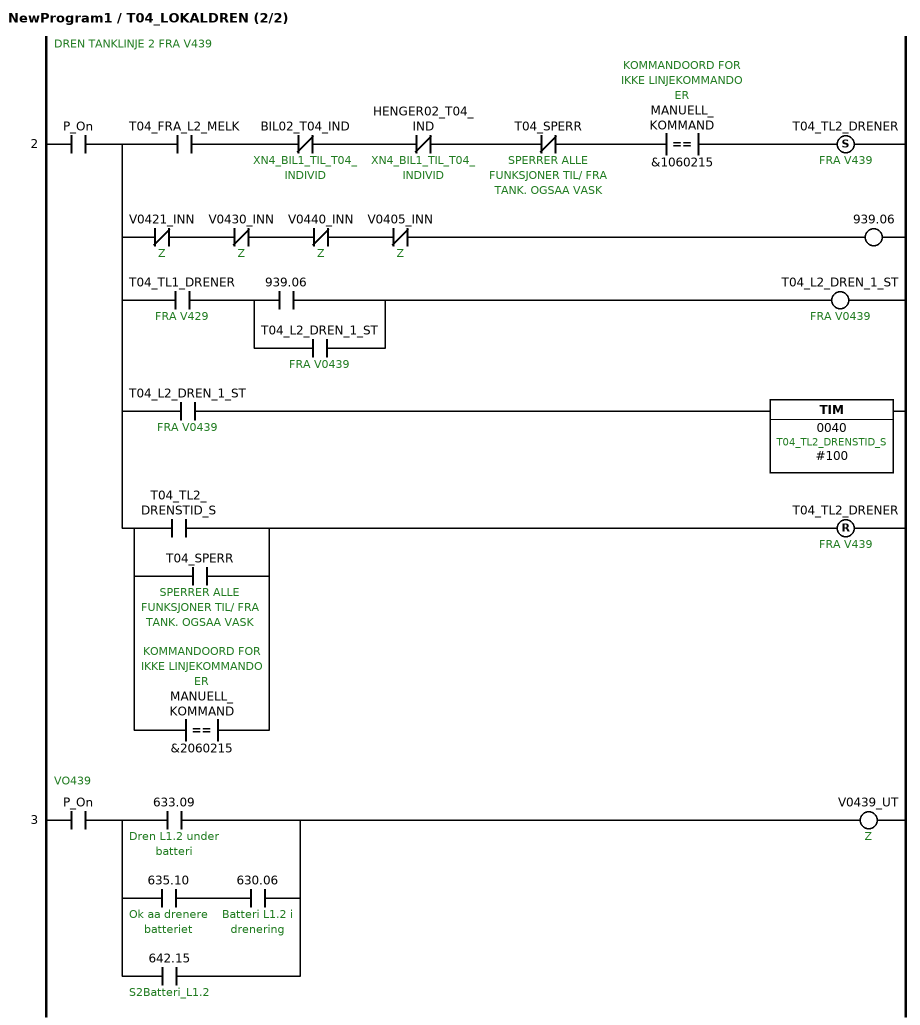
; rung 2: DREN TANKLINJE 2 FRA V439
LD P_On
OUT TR0
AND T04_FRA_L2_MELK
ANDNOT BIL02_T04_IND  ; XN4_BIL1_TIL_T04_INDIVID
ANDNOT HENGER02_T04_IND  ; XN4_BIL1_TIL_T04_INDIVID
ANDNOT T04_SPERR  ; SPERRER ALLE FUNKSJONER TIL/ FRA TANK. OGSAA VASK
AND=L(301) MANUELL_KOMMAND &1060215  ; KOMMANDOORD FOR IKKE LINJEKOMMANDOER
SET T04_TL2_DRENER  ; FRA V439
LD TR0
ANDNOT V0421_INN  ; Z
ANDNOT V0430_INN  ; Z
ANDNOT V0440_INN  ; Z
ANDNOT V0405_INN  ; Z
OUT 939.06
LD TR0
AND T04_TL1_DRENER  ; FRA V429
LD 939.06
OR T04_L2_DREN_1_ST  ; FRA V0439
ANDLD
OUT T04_L2_DREN_1_ST  ; FRA V0439
LD TR0
AND T04_L2_DREN_1_ST  ; FRA V0439
TIM 0040 #100  ; T04_TL2_DRENSTID_S
LD TR0
LD T04_TL2_DRENSTID_S
OR T04_SPERR  ; SPERRER ALLE FUNKSJONER TIL/ FRA TANK. OGSAA VASK
OR=L(301) MANUELL_KOMMAND &2060215  ; KOMMANDOORD FOR IKKE LINJEKOMMANDOER
ANDLD
RSET T04_TL2_DRENER  ; FRA V439
; rung 3: VO439
LD P_On
LD 633.09  ; Dren L1.2 under batteri
LD 635.10  ; Ok aa drenere batteriet
AND 630.06  ; Batteri L1.2 i drenering
ORLD
OR 642.15  ; S2Batteri_L1.2
ANDLD
OUT V0439_UT  ; Z
; rung 4: Ingen_kommentar_funnet

### Section T04_TEMP_NIVÅ

